FUNCTION_BLOCK MyPou
VAR_INPUT
END_VAR
VAR_OUTPUT
END_VAR
VAR
END_VAR

END_FUNCTION_BLOCK

(* stored: Version 1.1.0.1, ProductVersion 3.1.4024.13
   POU MyPou: Id {5326085c-492a-42b3-8a35-1c88a6f97b36}, SpecialFunc None *)
